FUNCTION_BLOCK FB_FMS205_F6Prueba_SFC EXTENDS FB_ControllerBase_SFC
VAR_INPUT
	FinCiclo : BOOL;
END_VAR

VAR_IN_OUT
	Alime			: FB_Alimentador;
	Carga		 	: FB_PickAndPlace;
	Medid			: FB_MedidorTapa;
	Induc		 	: FB_CaptadorInductivo;
	Fotoe			: FB_DetectorFotoelectrico;
	Evacu		 	: FB_Evacuador;
	Desca			: FB_PickAndPlace;
	Plato			: FB_PlatoDivisor;
	Cinta			: FB_Cinta;
END_VAR

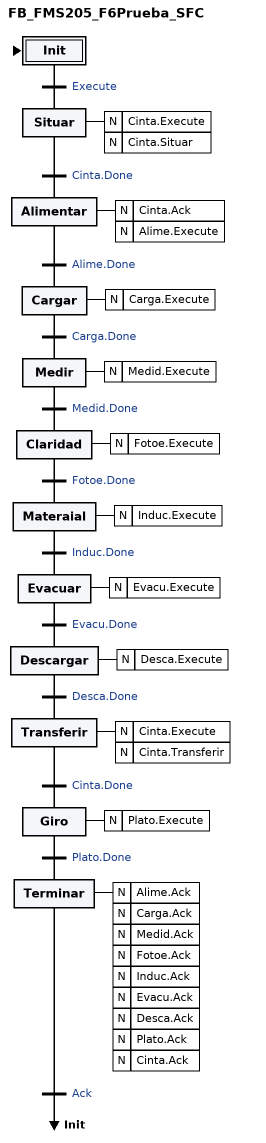
INITIAL_STEP Init:
END_STEP
TRANSITION FROM Init TO Situar
    := Execute;
END_TRANSITION
STEP Situar:
    Cinta.Execute(N);
    Cinta.Situar(N);
END_STEP
TRANSITION FROM Situar TO Alimentar
    := Cinta.Done;
END_TRANSITION
STEP Alimentar:
    Cinta.Ack(N);
    Alime.Execute(N);
END_STEP
TRANSITION FROM Alimentar TO Cargar
    := Alime.Done;
END_TRANSITION
STEP Cargar:
    Carga.Execute(N);
END_STEP
TRANSITION FROM Cargar TO Medir
    := Carga.Done;
END_TRANSITION
STEP Medir:
    Medid.Execute(N);
END_STEP
TRANSITION FROM Medir TO Claridad
    := Medid.Done;
END_TRANSITION
STEP Claridad:
    Fotoe.Execute(N);
END_STEP
TRANSITION FROM Claridad TO Materaial
    := Fotoe.Done;
END_TRANSITION
STEP Materaial:
    Induc.Execute(N);
END_STEP
TRANSITION FROM Materaial TO Evacuar
    := Induc.Done;
END_TRANSITION
STEP Evacuar:
    Evacu.Execute(N);
END_STEP
TRANSITION FROM Evacuar TO Descargar
    := Evacu.Done;
END_TRANSITION
STEP Descargar:
    Desca.Execute(N);
END_STEP
TRANSITION FROM Descargar TO Transferir
    := Desca.Done;
END_TRANSITION
STEP Transferir:
    Cinta.Execute(N);
    Cinta.Transferir(N);
END_STEP
TRANSITION FROM Transferir TO Giro
    := Cinta.Done;
END_TRANSITION
STEP Giro:
    Plato.Execute(N);
END_STEP
TRANSITION FROM Giro TO Terminar
    := Plato.Done;
END_TRANSITION
STEP Terminar:
    Alime.Ack(N);
    Carga.Ack(N);
    Medid.Ack(N);
    Fotoe.Ack(N);
    Induc.Ack(N);
    Evacu.Ack(N);
    Desca.Ack(N);
    Plato.Ack(N);
    Cinta.Ack(N);
END_STEP
TRANSITION FROM Terminar TO Init
    := Ack;
END_TRANSITION

END_FUNCTION_BLOCK

(* stored: Version 1.1.0.1, ProductVersion 3.1.4024.11
   POU FB_FMS205_F6Prueba_SFC: Id {a81c472c-1220-4b76-860b-f7f6b111694f}, SpecialFunc None *)
